// TIA Portal V20 export
ORGANIZATION_BLOCK "Main"   // OB1, LAD, ProgramCycle
TITLE = "Main Program Sweep (Cycle)"
{ S7_Optimized_Access := 'TRUE' }
// stored: SetENOAutomatically false
   VAR_INPUT
      Initial_Call : Bool;   // Initial call of this OB
      Remanence : Bool;   // =True, if remanent data are available
   END_VAR
BEGIN

REGION Network 1: CALL - Main machine modules (Not used)
   // Call of the application's main machine functions (NOT used)
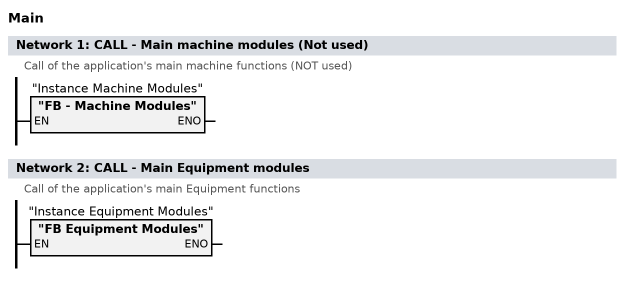
   RUNG wire#powerrail
      "Instance Machine Modules"()
   END_RUNG
   // the same network as SCL:
   "Instance Machine Modules"();   // "FB - Machine Modules"
END_REGION

REGION Network 2: CALL - Main Equipment modules
   // Call of the application's main Equipment functions
   RUNG wire#powerrail
      "Instance Equipment Modules"()
   END_RUNG
   // the same network as SCL:
   "Instance Equipment Modules"();   // "FB Equipment Modules"
END_REGION
END_ORGANIZATION_BLOCK
